// TIA Portal V20 export
// export: Created 2025-12-01T14:56:58.036077Z, ExportSetting None, DisplayName Totally Integrated Automation Portal, DisplayVersion V20 Update 3, DisplayName TIA Portal Openness, DisplayVersion V20 Update 3, DisplayName TIA Portal Version Control Interface, DisplayVersion V20 Update 3, DisplayName STEP 7 Professional, DisplayVersion V20 Update 3, DisplayName STEP 7 Safety, DisplayVersion V20 Update 2, DisplayName WinCC Basic/Comfort/Advanced, DisplayVersion V20 Update 3, DisplayName WinCC Professional, DisplayVersion V20 Update 3, DisplayName WinCC Unified, DisplayVersion V20 Update 3
FUNCTION_BLOCK "FB85_GALIBO_5Alturas"   // FB85, LAD
TITLE = Galibo de 5 Alturas (2023)
{ S7_Optimized_Access := 'FALSE' }
AUTHOR : GALIBO
NAME : 20140101
VERSION : 3.0
// stored: AutoNumber false, SetENOAutomatically false
   VAR_INPUT
      Mesa : UInt;
      NumGalibo : UInt;
      pHs_ALT_1 : Bool;
      pHs_ALT_2 : Bool;
      pHs_ALT_3 : Bool;
      pHs_ALT_4 : Bool;
      pHs_ERR_ALT : Bool;
      HabilitarLectura : Bool;
      PermisoLectura : Bool;
      Rearmar_ConMesaLibre : Bool;
   END_VAR
   VAR_OUTPUT
      Baliza : Bool;
      ErrorAltura : Bool;
      FinLectura : Bool;
   END_VAR
   VAR
      GAL_ET00 : Bool;
      GAL_ET01 : Bool;
      GAL_ET02 : Bool;
      GAL_ET03 : Bool;
      pHsGalibo_OK { ExternalAccessible := 'False'; ExternalVisible := 'False'; ExternalWritable := 'False'} : Bool;
      LeerAltura : Bool;
      Altura_NOOK : Bool;
      Altura_OK_1 : Bool;
      Altura_OK_2 : Bool;
      Altura_OK_3 : Bool;
      Altura_OK_4 : Bool;
      Altura_OK_5 : Bool;
      CodigoAltura : SInt;
      MemoCodigo : Word;
      STAT_Baliza_Galibo : Bool;
   END_VAR
   VAR_TEMP
      EstadoZona : "EstadoZona";
      EstadoVI : "EstadosMesa";
   END_VAR
   VAR_TEMP   // added for the SCL form of the ladder/FBD networks
      _w1 : Bool;
   END_VAR
BEGIN

REGION Network 1: INICIALIZAR - Recoger las Variables de Estado de la Mesa
   // Se recoge - Estado_CBx
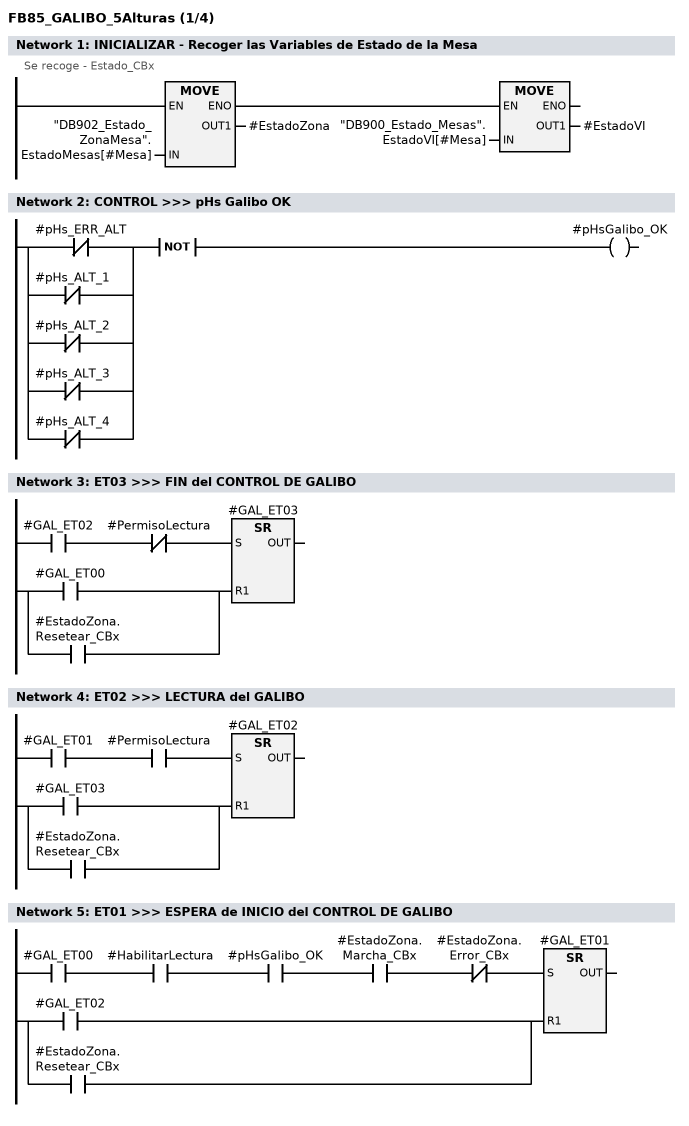
   RUNG wire#powerrail
      Move(in := "DB902_Estado_ZonaMesa".EstadoMesas[#Mesa], out1 => #EstadoZona)
      Move(in := "DB900_Estado_Mesas".EstadoVI[#Mesa], out1 => #EstadoVI)
   END_RUNG
   // the same network as SCL:
   #EstadoZona := "DB902_Estado_ZonaMesa".EstadoMesas[#Mesa];
   #EstadoVI := "DB900_Estado_Mesas".EstadoVI[#Mesa];
END_REGION

REGION Network 2: CONTROL >>> pHs Galibo OK
   RUNG wire#powerrail
      I_Contact( #pHs_ERR_ALT )
      wire#w1
      Not()
      Coil( #pHsGalibo_OK )
   END_RUNG
   RUNG wire#powerrail
      I_Contact( #pHs_ALT_1 )
   END_RUNG wire#w1
   RUNG wire#powerrail
      I_Contact( #pHs_ALT_2 )
   END_RUNG wire#w1
   RUNG wire#powerrail
      I_Contact( #pHs_ALT_3 )
   END_RUNG wire#w1
   RUNG wire#powerrail
      I_Contact( #pHs_ALT_4 )
   END_RUNG wire#w1
   // the same network as SCL:
   #pHsGalibo_OK := NOT (NOT #pHs_ERR_ALT OR NOT #pHs_ALT_1 OR NOT #pHs_ALT_2 OR NOT #pHs_ALT_3 OR NOT #pHs_ALT_4);
END_REGION

REGION Network 3: ET03 >>> FIN del CONTROL DE GALIBO
   RUNG wire#powerrail
      Contact( #GAL_ET02 )
      I_Contact( #PermisoLectura )
      S_SR(operand := #GAL_ET03, r1 := wire#w1)
   END_RUNG
   RUNG wire#powerrail
      Contact( #GAL_ET00 )
   END_RUNG wire#w1
   RUNG wire#powerrail
      Contact( #EstadoZona.Resetear_CBx )
   END_RUNG wire#w1
   // the same network as SCL:
   IF #GAL_ET02 AND NOT #PermisoLectura THEN
       #GAL_ET03 := TRUE;   // SR flip-flop
   END_IF;
   IF #GAL_ET00 OR #EstadoZona.Resetear_CBx THEN #GAL_ET03 := FALSE; END_IF;
END_REGION

REGION Network 4: ET02 >>> LECTURA del GALIBO
   RUNG wire#powerrail
      Contact( #GAL_ET01 )
      Contact( #PermisoLectura )
      S_SR(operand := #GAL_ET02, r1 := wire#w1)
   END_RUNG
   RUNG wire#powerrail
      Contact( #GAL_ET03 )
   END_RUNG wire#w1
   RUNG wire#powerrail
      Contact( #EstadoZona.Resetear_CBx )
   END_RUNG wire#w1
   // the same network as SCL:
   IF #GAL_ET01 AND #PermisoLectura THEN
       #GAL_ET02 := TRUE;   // SR flip-flop
   END_IF;
   IF #GAL_ET03 OR #EstadoZona.Resetear_CBx THEN #GAL_ET02 := FALSE; END_IF;
END_REGION

REGION Network 5: ET01 >>> ESPERA de INICIO del CONTROL DE GALIBO
   RUNG wire#powerrail
      Contact( #GAL_ET00 )
      Contact( #HabilitarLectura )
      Contact( #pHsGalibo_OK )
      Contact( #EstadoZona.Marcha_CBx )
      I_Contact( #EstadoZona.Error_CBx )
      S_SR(operand := #GAL_ET01, r1 := wire#w1)
   END_RUNG
   RUNG wire#powerrail
      Contact( #GAL_ET02 )
   END_RUNG wire#w1
   RUNG wire#powerrail
      Contact( #EstadoZona.Resetear_CBx )
   END_RUNG wire#w1
   // the same network as SCL:
   IF #GAL_ET00 AND #HabilitarLectura AND #pHsGalibo_OK AND #EstadoZona.Marcha_CBx AND NOT #EstadoZona.Error_CBx THEN
       #GAL_ET01 := TRUE;   // SR flip-flop
   END_IF;
   IF #GAL_ET02 OR #EstadoZona.Resetear_CBx THEN #GAL_ET01 := FALSE; END_IF;
END_REGION

REGION Network 6: ET00 >>> INICIO
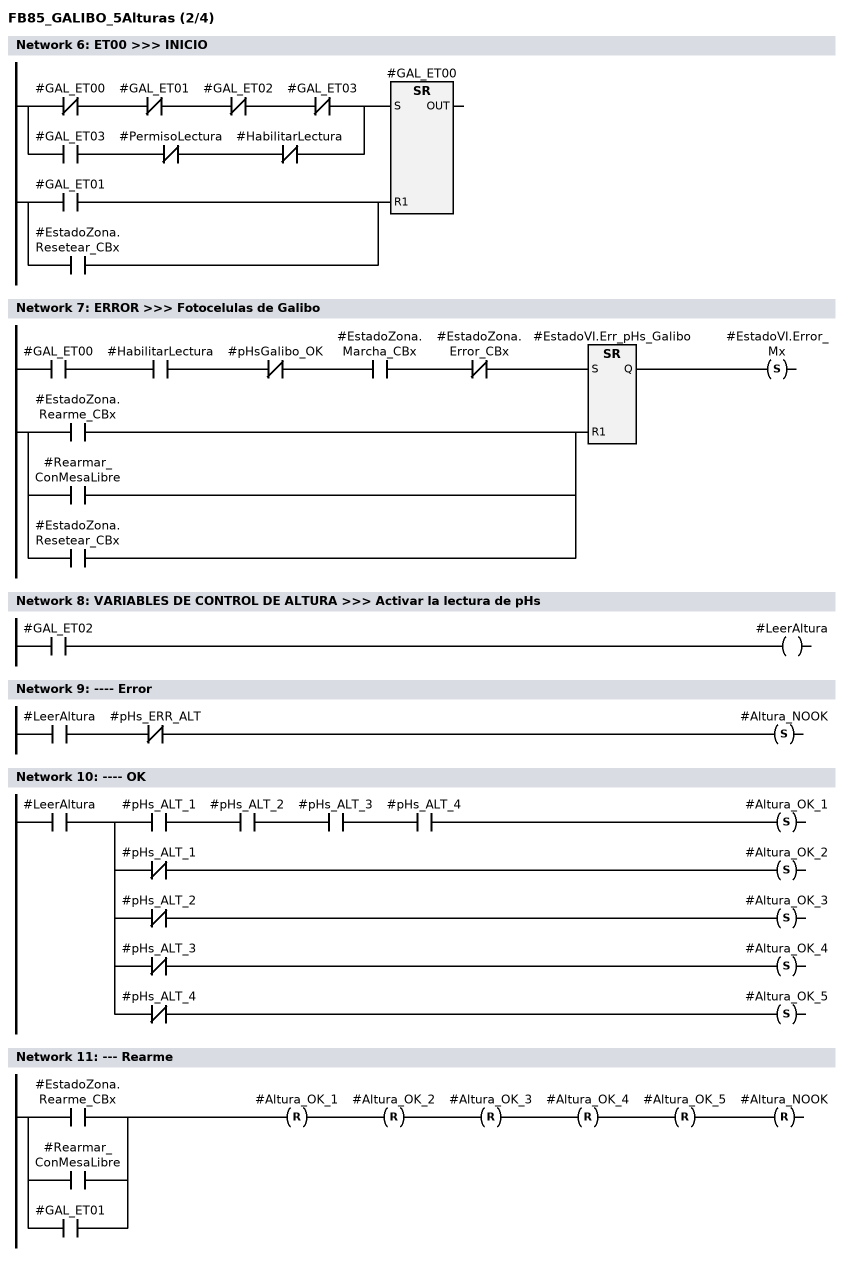
   RUNG wire#powerrail
      I_Contact( #GAL_ET00 )
      I_Contact( #GAL_ET01 )
      I_Contact( #GAL_ET02 )
      I_Contact( #GAL_ET03 )
      wire#w1
      S_SR(operand := #GAL_ET00, r1 := wire#w2)
   END_RUNG
   RUNG wire#powerrail
      Contact( #GAL_ET03 )
      I_Contact( #PermisoLectura )
      I_Contact( #HabilitarLectura )
   END_RUNG wire#w1
   RUNG wire#powerrail
      Contact( #GAL_ET01 )
   END_RUNG wire#w2
   RUNG wire#powerrail
      Contact( #EstadoZona.Resetear_CBx )
   END_RUNG wire#w2
   // the same network as SCL:
   IF (NOT #GAL_ET00 AND NOT #GAL_ET01 AND NOT #GAL_ET02 AND NOT #GAL_ET03) OR (#GAL_ET03 AND NOT #PermisoLectura AND NOT #HabilitarLectura) THEN
       #GAL_ET00 := TRUE;   // SR flip-flop
   END_IF;
   IF #GAL_ET01 OR #EstadoZona.Resetear_CBx THEN #GAL_ET00 := FALSE; END_IF;
END_REGION

REGION Network 7: ERROR >>> Fotocelulas de Galibo
   RUNG wire#powerrail
      Contact( #GAL_ET00 )
      Contact( #HabilitarLectura )
      I_Contact( #pHsGalibo_OK )
      Contact( #EstadoZona.Marcha_CBx )
      I_Contact( #EstadoZona.Error_CBx )
      S_SR(operand := #EstadoVI.Err_pHs_Galibo, r1 := wire#w1)
      S_Coil( #EstadoVI.Error_Mx )
   END_RUNG
   RUNG wire#powerrail
      Contact( #EstadoZona.Rearme_CBx )
   END_RUNG wire#w1
   RUNG wire#powerrail
      Contact( #Rearmar_ConMesaLibre )
   END_RUNG wire#w1
   RUNG wire#powerrail
      Contact( #EstadoZona.Resetear_CBx )
   END_RUNG wire#w1
   // the same network as SCL:
   IF #GAL_ET00 AND #HabilitarLectura AND NOT #pHsGalibo_OK AND #EstadoZona.Marcha_CBx AND NOT #EstadoZona.Error_CBx THEN
       #EstadoVI.Err_pHs_Galibo := TRUE;   // SR flip-flop
   END_IF;
   IF #EstadoZona.Rearme_CBx OR #Rearmar_ConMesaLibre OR #EstadoZona.Resetear_CBx THEN
       #EstadoVI.Err_pHs_Galibo := FALSE;
   END_IF;
   IF #EstadoVI.Err_pHs_Galibo THEN #EstadoVI.Error_Mx := TRUE; END_IF;
END_REGION

REGION Network 8: VARIABLES DE CONTROL DE ALTURA >>> Activar la lectura de pHs
   RUNG wire#powerrail
      Contact( #GAL_ET02 )
      Coil( #LeerAltura )
   END_RUNG
   // the same network as SCL:
   #LeerAltura := #GAL_ET02;
END_REGION

REGION Network 9: ---- Error
   RUNG wire#powerrail
      Contact( #LeerAltura )
      I_Contact( #pHs_ERR_ALT )
      S_Coil( #Altura_NOOK )
   END_RUNG
   // the same network as SCL:
   IF #LeerAltura AND NOT #pHs_ERR_ALT THEN #Altura_NOOK := TRUE; END_IF;
END_REGION

REGION Network 10: ---- OK
   RUNG wire#powerrail
      Contact( #LeerAltura )
      wire#w1
      Contact( #pHs_ALT_1 )
      Contact( #pHs_ALT_2 )
      Contact( #pHs_ALT_3 )
      Contact( #pHs_ALT_4 )
      S_Coil( #Altura_OK_1 )
   END_RUNG
   RUNG wire#w1
      I_Contact( #pHs_ALT_1 )
      S_Coil( #Altura_OK_2 )
   END_RUNG
   RUNG wire#w1
      I_Contact( #pHs_ALT_2 )
      S_Coil( #Altura_OK_3 )
   END_RUNG
   RUNG wire#w1
      I_Contact( #pHs_ALT_3 )
      S_Coil( #Altura_OK_4 )
   END_RUNG
   RUNG wire#w1
      I_Contact( #pHs_ALT_4 )
      S_Coil( #Altura_OK_5 )
   END_RUNG
   // the same network as SCL:
   IF #LeerAltura AND #pHs_ALT_1 AND #pHs_ALT_2 AND #pHs_ALT_3 AND #pHs_ALT_4 THEN
       #Altura_OK_1 := TRUE;
   END_IF;
   IF #LeerAltura AND NOT #pHs_ALT_1 THEN #Altura_OK_2 := TRUE; END_IF;
   IF #LeerAltura AND NOT #pHs_ALT_2 THEN #Altura_OK_3 := TRUE; END_IF;
   IF #LeerAltura AND NOT #pHs_ALT_3 THEN #Altura_OK_4 := TRUE; END_IF;
   IF #LeerAltura AND NOT #pHs_ALT_4 THEN #Altura_OK_5 := TRUE; END_IF;
END_REGION

REGION Network 11: --- Rearme
   RUNG wire#powerrail
      Contact( #EstadoZona.Rearme_CBx )
      wire#w1
      R_Coil( #Altura_OK_1 )
      R_Coil( #Altura_OK_2 )
      R_Coil( #Altura_OK_3 )
      R_Coil( #Altura_OK_4 )
      R_Coil( #Altura_OK_5 )
      R_Coil( #Altura_NOOK )
   END_RUNG
   RUNG wire#powerrail
      Contact( #Rearmar_ConMesaLibre )
   END_RUNG wire#w1
   RUNG wire#powerrail
      Contact( #GAL_ET01 )
   END_RUNG wire#w1
   // the same network as SCL:
   IF #EstadoZona.Rearme_CBx OR #Rearmar_ConMesaLibre OR #GAL_ET01 THEN
       #Altura_OK_1 := FALSE;
       #Altura_OK_2 := FALSE;
       #Altura_OK_3 := FALSE;
       #Altura_OK_4 := FALSE;
       #Altura_OK_5 := FALSE;
       #Altura_NOOK := FALSE;
   END_IF;
END_REGION

REGION Network 12: CODIFICACION DEL GALIBO >>> Inicialiar
   // Por Defecto >>> Sin realizar lectura
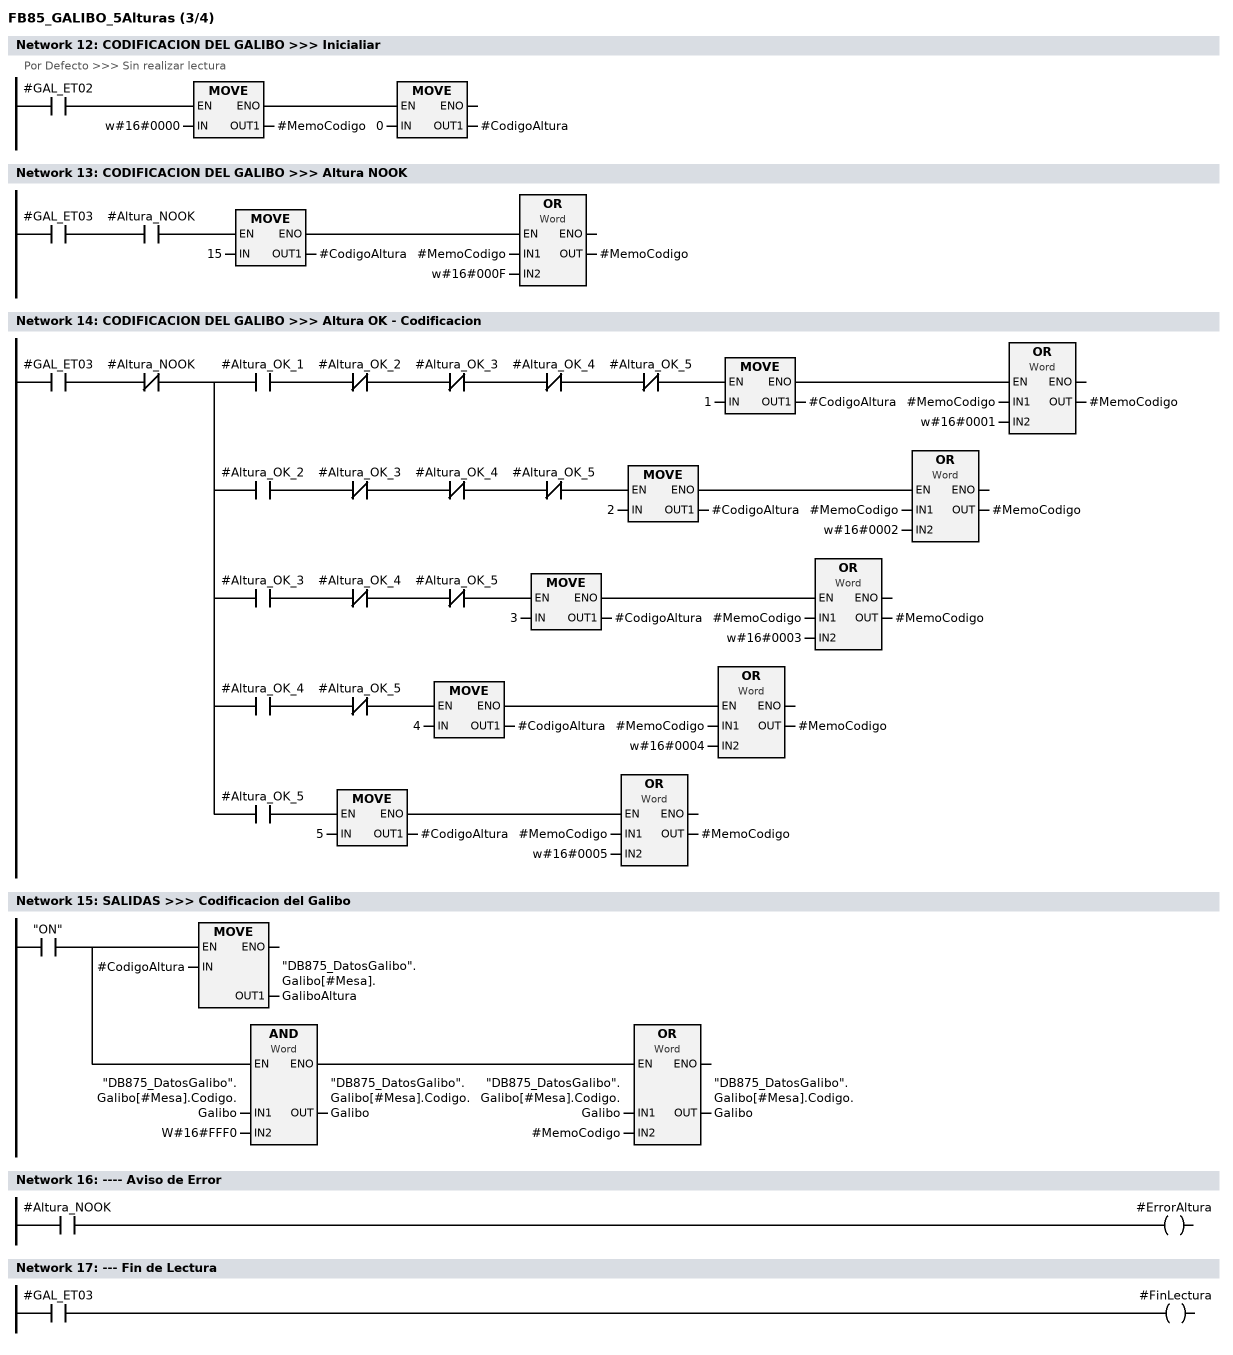
   RUNG wire#powerrail
      Contact( #GAL_ET02 )
      { S7_GenerateENO := "TRUE" } Move(in := w#16#0000, out1 => #MemoCodigo)
      { S7_GenerateENO := "TRUE" } Move(in := 0, out1 => #CodigoAltura)
   END_RUNG
   // the same network as SCL:
   // ENO of a box is taken as its EN; it also drops when the box reports an error
   IF #GAL_ET02 THEN
       #MemoCodigo := w#16#0000;
       #CodigoAltura := 0;
   END_IF;
END_REGION

REGION Network 13: CODIFICACION DEL GALIBO >>> Altura NOOK
   // ENO of a box is taken as its EN; it also drops when the box reports an error
   IF #GAL_ET03 AND #Altura_NOOK THEN
       #CodigoAltura := 15;
       #MemoCodigo := #MemoCodigo OR w#16#000F;
   END_IF;
END_REGION

REGION Network 14: CODIFICACION DEL GALIBO >>> Altura OK - Codificacion
   // ENO of a box is taken as its EN; it also drops when the box reports an error
   #_w1 := #GAL_ET03 AND NOT #Altura_NOOK;
   IF #_w1 AND #Altura_OK_1 AND NOT #Altura_OK_2 AND NOT #Altura_OK_3 AND NOT #Altura_OK_4 AND NOT #Altura_OK_5 THEN
       #CodigoAltura := 1;
       #MemoCodigo := #MemoCodigo OR w#16#0001;
   END_IF;
   IF #_w1 AND #Altura_OK_2 AND NOT #Altura_OK_3 AND NOT #Altura_OK_4 AND NOT #Altura_OK_5 THEN
       #CodigoAltura := 2;
       #MemoCodigo := #MemoCodigo OR w#16#0002;
   END_IF;
   IF #_w1 AND #Altura_OK_3 AND NOT #Altura_OK_4 AND NOT #Altura_OK_5 THEN
       #CodigoAltura := 3;
       #MemoCodigo := #MemoCodigo OR w#16#0003;
   END_IF;
   IF #_w1 AND #Altura_OK_4 AND NOT #Altura_OK_5 THEN
       #CodigoAltura := 4;
       #MemoCodigo := #MemoCodigo OR w#16#0004;
   END_IF;
   IF #_w1 AND #Altura_OK_5 THEN
       #CodigoAltura := 5;
       #MemoCodigo := #MemoCodigo OR w#16#0005;
   END_IF;
END_REGION

REGION Network 15: SALIDAS >>> Codificacion del Galibo
   IF "ON" THEN
       "DB875_DatosGalibo".Galibo[#Mesa].GaliboAltura := #CodigoAltura;
       "DB875_DatosGalibo".Galibo[#Mesa].Codigo.Galibo := "DB875_DatosGalibo".Galibo[#Mesa].Codigo.Galibo AND W#16#FFF0;
       "DB875_DatosGalibo".Galibo[#Mesa].Codigo.Galibo := "DB875_DatosGalibo".Galibo[#Mesa].Codigo.Galibo OR #MemoCodigo;
   END_IF;
END_REGION

REGION Network 16: ---- Aviso de Error
   RUNG wire#powerrail
      Contact( #Altura_NOOK )
      Coil( #ErrorAltura )
   END_RUNG
   // the same network as SCL:
   #ErrorAltura := #Altura_NOOK;
END_REGION

REGION Network 17: --- Fin de Lectura
   RUNG wire#powerrail
      Contact( #GAL_ET03 )
      Coil( #FinLectura )
   END_RUNG
   // the same network as SCL:
   #FinLectura := #GAL_ET03;
END_REGION

REGION Network 18: SALIDAS >>> BALIZA
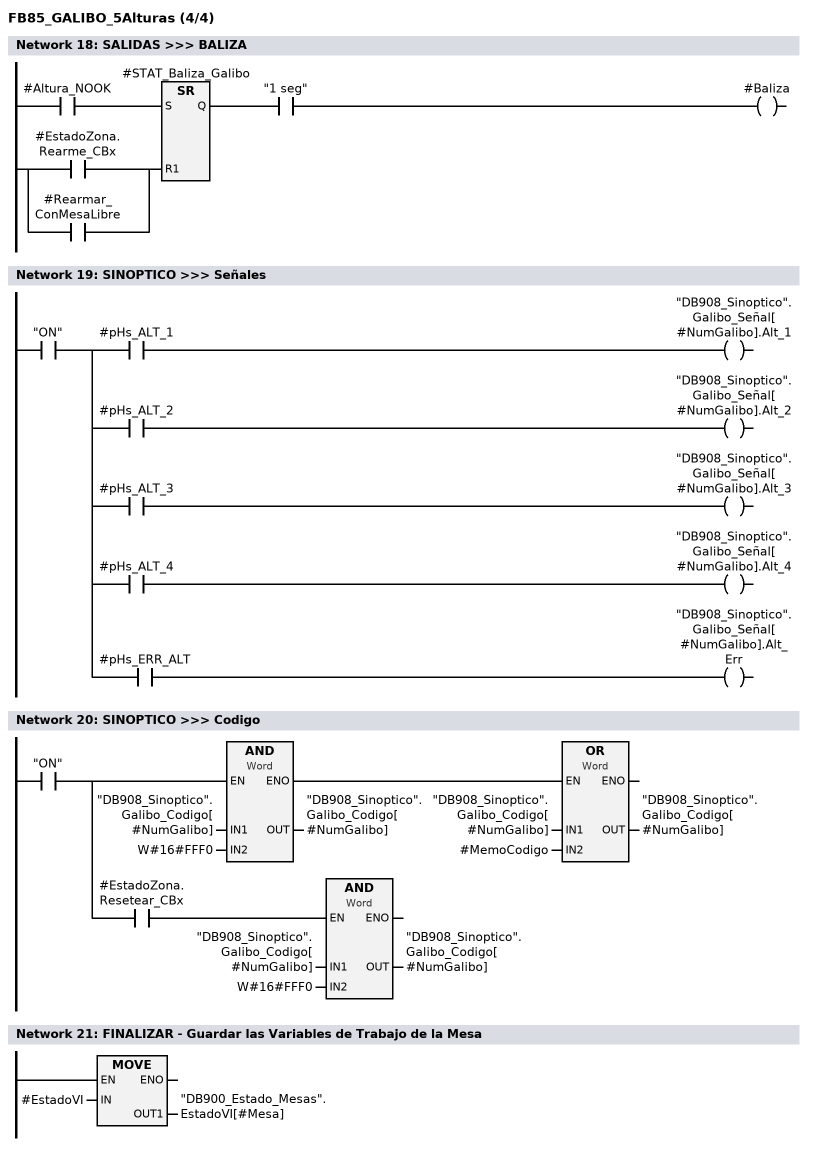
   RUNG wire#powerrail
      Contact( #Altura_NOOK )
      S_SR(operand := #STAT_Baliza_Galibo, r1 := wire#w1)
      Contact( "1 seg" )
      Coil( #Baliza )
   END_RUNG
   RUNG wire#powerrail
      Contact( #EstadoZona.Rearme_CBx )
   END_RUNG wire#w1
   RUNG wire#powerrail
      Contact( #Rearmar_ConMesaLibre )
   END_RUNG wire#w1
   // the same network as SCL:
   IF #Altura_NOOK THEN
       #STAT_Baliza_Galibo := TRUE;   // SR flip-flop
   END_IF;
   IF #EstadoZona.Rearme_CBx OR #Rearmar_ConMesaLibre THEN #STAT_Baliza_Galibo := FALSE; END_IF;
   #Baliza := #STAT_Baliza_Galibo AND "1 seg";
END_REGION

REGION Network 19: SINOPTICO >>> Señales
   RUNG wire#powerrail
      Contact( "ON" )
      wire#w1
      Contact( #pHs_ALT_1 )
      Coil( "DB908_Sinoptico".Galibo_Señal[#NumGalibo].Alt_1 )
   END_RUNG
   RUNG wire#w1
      Contact( #pHs_ALT_2 )
      Coil( "DB908_Sinoptico".Galibo_Señal[#NumGalibo].Alt_2 )
   END_RUNG
   RUNG wire#w1
      Contact( #pHs_ALT_3 )
      Coil( "DB908_Sinoptico".Galibo_Señal[#NumGalibo].Alt_3 )
   END_RUNG
   RUNG wire#w1
      Contact( #pHs_ALT_4 )
      Coil( "DB908_Sinoptico".Galibo_Señal[#NumGalibo].Alt_4 )
   END_RUNG
   RUNG wire#w1
      Contact( #pHs_ERR_ALT )
      Coil( "DB908_Sinoptico".Galibo_Señal[#NumGalibo].Alt_Err )
   END_RUNG
   // the same network as SCL:
   "DB908_Sinoptico".Galibo_Señal[#NumGalibo].Alt_1 := "ON" AND #pHs_ALT_1;
   "DB908_Sinoptico".Galibo_Señal[#NumGalibo].Alt_2 := "ON" AND #pHs_ALT_2;
   "DB908_Sinoptico".Galibo_Señal[#NumGalibo].Alt_3 := "ON" AND #pHs_ALT_3;
   "DB908_Sinoptico".Galibo_Señal[#NumGalibo].Alt_4 := "ON" AND #pHs_ALT_4;
   "DB908_Sinoptico".Galibo_Señal[#NumGalibo].Alt_Err := "ON" AND #pHs_ERR_ALT;
END_REGION

REGION Network 20: SINOPTICO >>> Codigo
   IF "ON" THEN
       "DB908_Sinoptico".Galibo_Codigo[#NumGalibo] := "DB908_Sinoptico".Galibo_Codigo[#NumGalibo] AND W#16#FFF0;
       "DB908_Sinoptico".Galibo_Codigo[#NumGalibo] := "DB908_Sinoptico".Galibo_Codigo[#NumGalibo] OR #MemoCodigo;
   END_IF;
   IF "ON" AND #EstadoZona.Resetear_CBx THEN
       "DB908_Sinoptico".Galibo_Codigo[#NumGalibo] := "DB908_Sinoptico".Galibo_Codigo[#NumGalibo] AND W#16#FFF0;
   END_IF;
END_REGION

REGION Network 21: FINALIZAR - Guardar las Variables de Trabajo de la Mesa
   RUNG wire#powerrail
      Move(in := #EstadoVI, out1 => "DB900_Estado_Mesas".EstadoVI[#Mesa])
   END_RUNG
   // the same network as SCL:
   "DB900_Estado_Mesas".EstadoVI[#Mesa] := #EstadoVI;
END_REGION
END_FUNCTION_BLOCK
